FUNCTION cycl_change : INT
VAR_INPUT
	i_cycle_int: INT;
	i_increment: INT;
END_VAR
VAR

END_VAR



i_cycle_int := i_cycle_int + i_increment;
cycl_change := i_cycle_int;

END_FUNCTION

(* stored: Version 1.1.0.1, ProductVersion 3.1.4022.7
   POU cycl_change: Id {26e569ac-8463-4eef-bb66-3bbe3f6745ca}, SpecialFunc None *)
